{attribute 'TcGenerated'}
// This function has been automatically generated from the project information.
VAR_GLOBAL CONSTANT
    {attribute 'const_non_replaced'}
    {attribute 'linkalways'}
    stLibVersion_lcls_plc_tmo_optics : ST_LibVersion := (iMajor := 3, iMinor := 1, iBuild := 0, iRevision := 0, sVersion := '3.1.0');
END_VAR

(* stored: Version 1.1.0.1, ProductVersion 3.1.4022.18
   GVL Global_Version: Id 8dec1fc8-6ae3-4489-bd6b-2d3996940111 *)
